PROGRAM MAIN
VAR
	FbMotion1: Fb_Motion;
	FbMotion2: Fb_Motion;
	nState: INT;
	bButon: BOOL;
	T1: TON;
	T2: TON;
	T3: TON;
	bResetButon	:	BOOL;
	rtrig1: R_TRIG;
	bCounter: BOOL;
	nCounter: INT;
	sMsgInfo: STRING;
	sMsgVelo: STRING;
	sMsgPosition: STRING;
	fPositionVisu: LREAL;
END_VAR



ACT_Motion();
ACT_Visu();







FbMotion1(Axis:=GVL_Axis.Axis1 , stAxis:=GVL_Axis.stAxis1 );
//FbMotion2(Axis:=GVL_Axis.Axis2 , stAxis:=GVL_Axis.stAxis2 );

ACTION ACT_Motion:


rtrig1(CLK:=bCounter , Q=> );


CASE nState OF
	



	0:
	
		IF bButon THEN
			
		GVL_Axis.stAxis1.IN.bPowerEnable	:=	TRUE;
		GVL_Axis.stAxis1.IN.fOverride	:=	100.0;
		GVL_Axis.stAxis1.IN.bStop	:=	FALSE;	
		GVL_Axis.stAxis1.IN.bMoveAbs	:=	FALSE;
		nState := 1;
		
		END_IF
	
		
	1:
		IF	bButon	
		AND NOT GVL_Axis.stAxis1.OUT.bPowerErr
		AND NOT GVL_Axis.stAxis1.OUT.bStopActive 
		AND GVL_Axis.stAxis1.OUT.bPowerEnabled THEN
		
			nState := 10;
			
		END_IF
	
	
	10:
		
		GVL_Axis.stAxis1.IN.fPosition	:=	5000;
		GVL_Axis.stAxis1.IN.fVelocity	:=	650;
		
		GVL_Axis.stAxis1.IN.bMoveAbs	:=	TRUE;
		
		IF GVL_Axis.stAxis1.OUT.bMoveAbsBusy 
		AND NOT GVL_Axis.stAxis1.OUT.bMoveAbsErr	THEN
			
			nState := 20;

		ELSIF 	GVL_Axis.stAxis1.OUT.bMoveAbsErr 
		OR GVL_Axis.stAxis1.OUT.bPowerErr THEN
			
			nState := 999;
		
		END_IF
		
	20:
		sMsgInfo	:=	'Sistem Belirtilen Pozisyona Hareket Etmekte';
		
		IF GVL_Axis.stAxis1.OUT.bMoveAbsDone
		AND NOT GVL_Axis.stAxis1.OUT.bMoveAbsErr THEN
		
			GVL_Axis.stAxis1.IN.bMoveAbs	:=	FALSE;	
			nState := 30;
		
		ELSIF 	GVL_Axis.stAxis1.OUT.bMoveAbsErr 
		OR GVL_Axis.stAxis1.OUT.bPowerErr THEN
			
		nState := 999;
					
		END_IF
		
	
	30:
		
		sMsgInfo	:=	CONCAT(STR1:=TIME_TO_STRING(T1.ET) , STR2:='süredir bekleniyor.' );
	
		T1(IN:= TRUE, PT:=T#5S);
		
		IF T1.Q THEN
			nState := 40;
			T1(IN:= FALSE);
		END_IF
	
	40:
	
	
		GVL_Axis.stAxis1.IN.fPosition	:=	10000;
		GVL_Axis.stAxis1.IN.fVelocity	:=	1000;
		
		GVL_Axis.stAxis1.IN.bMoveAbs	:=	TRUE;
		
		IF GVL_Axis.stAxis1.OUT.bMoveAbsBusy 
		AND NOT GVL_Axis.stAxis1.OUT.bMoveAbsErr	THEN
			
			nState := 50;

		ELSIF 	GVL_Axis.stAxis1.OUT.bMoveAbsErr 
		OR GVL_Axis.stAxis1.OUT.bPowerErr THEN
			
			nState := 999;
		
		END_IF
		
	50:
		sMsgInfo	:=	'Sistem Belirtilen Pozisyona Hareket Etmekte';

		IF GVL_Axis.stAxis1.OUT.bMoveAbsDone
		AND NOT GVL_Axis.stAxis1.OUT.bMoveAbsErr THEN
		
			GVL_Axis.stAxis1.IN.bMoveAbs	:=	FALSE;	
			nState := 60;
		
		ELSIF 	GVL_Axis.stAxis1.OUT.bMoveAbsErr 
		OR GVL_Axis.stAxis1.OUT.bPowerErr THEN
			
		nState := 999;
					
		END_IF
	
	
	60:
		sMsgInfo	:=	'Malzemeler Bekleniyor.';
		IF rtrig1.Q THEN
			nCounter := nCounter + 1;			
		END_IF
		IF nCounter >=6 THEN
			nCounter := 0;
			nState := 70;
		END_IF
		
	70:
		
		GVL_Axis.stAxis1.IN.fPosition	:=	0;
		GVL_Axis.stAxis1.IN.fVelocity	:=	2000;
		
		GVL_Axis.stAxis1.IN.bMoveAbs	:=	TRUE;
		
		IF GVL_Axis.stAxis1.OUT.bMoveAbsBusy 
		AND NOT GVL_Axis.stAxis1.OUT.bMoveAbsErr	THEN
			
			nState := 80;

		ELSIF 	GVL_Axis.stAxis1.OUT.bMoveAbsErr 
		OR GVL_Axis.stAxis1.OUT.bPowerErr THEN
			
			nState := 999;
		
		END_IF
	
	
	80:
		sMsgInfo	:=	'Başlangıç Pozisyonuna Dönülüyor.';
		
		IF GVL_Axis.stAxis1.OUT.bMoveAbsDone
		AND NOT GVL_Axis.stAxis1.OUT.bMoveAbsErr THEN
		
			GVL_Axis.stAxis1.IN.bMoveAbs	:=	FALSE;	
			nState := 90;
		
		ELSIF 	GVL_Axis.stAxis1.OUT.bMoveAbsErr 
		OR GVL_Axis.stAxis1.OUT.bPowerErr THEN
			
		nState := 999;
					
		END_IF
		
	90:
		T3(IN:= TRUE, PT:=T#3S);
		
		IF T3.Q THEN
			nState := 0;
			T3(IN:= FALSE);
		END_IF
	

		
		
	999:
		GVL_Axis.stAxis1.IN.bReset	:=	TRUE;
		
		IF NOT	GVL_Axis.stAxis1.OUT.bResetErr 
		AND GVL_Axis.stAxis1.OUT.bResetDone
		AND bResetButon THEN
	
			nState := 0;
		
		ELSIF	GVL_Axis.stAxis1.OUT.bResetErr THEN
			nState := 1000;
		END_IF
		
		
		
END_CASE



IF NOT bButon THEN
	

	sMsgInfo	:=	'Sistem Kapalı Durumda.';

	T1(IN:= FALSE);
	T2(IN:= FALSE);
	T3(IN:= FALSE);
	
	GVL_Axis.stAxis1.IN.bStop	:=	TRUE;
	
	IF GVL_Axis.stAxis1.OUT.bStopDone
	AND 	GVL_Axis.stAxis1.OUT.bStopActive
	AND NOT	GVL_Axis.stAxis1.OUT.bMoveAbsErr
	AND NOT GVL_Axis.stAxis1.OUT.bPowerErr	 THEN
	
			nState := 0;
		
			GVL_Axis.stAxis1.IN.bPowerEnable	:=	TRUE;
			GVL_Axis.stAxis1.IN.fOverride	:=	100.0;
			
			GVL_Axis.stAxis1.IN.bStop	:=	FALSE;	
	END_IF
	
END_IF
END_ACTION

ACTION ACT_Visu:


sMsgVelo		:=	REAL_TO_STRING(GVL_Axis.Axis1.NcToPlc.ActVelo);
sMsgPosition	:=	REAL_TO_STRING(GVL_Axis.Axis1.NcToPlc.ActPos);


fPositionVisu	:=	GVL_Axis.Axis1.NcToPlc.ActPos/10;
END_ACTION

END_PROGRAM

(* stored: Version 1.1.0.1, ProductVersion 3.1.4024.4
   POU MAIN: Id {1f8f76ba-55d4-404a-8c87-3d73e978cf49}, SpecialFunc None
   Action ACT_Motion: Id {875773c2-5290-4d02-a306-85f1c937bb1c}
   Action ACT_Visu: Id {07620e5b-0f8b-4cbb-9964-3c2cf1401821} *)
